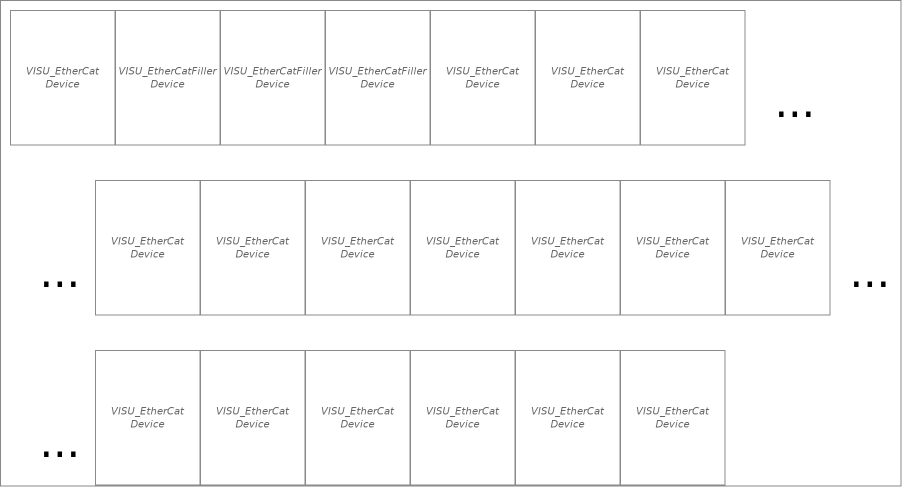
VISUALIZATION VISU_M1M2IO  // 902x487
VAR_IN_OUT
	ref : M1M2IO;
    widget : M1M2IOWidget;
END_VAR
    Frame (10,10 105x135)
        shows VISU_EtherCatDevice(device := ref.parts.COU, widget := widget.COU)
    Frame (535,10 105x135)
        shows VISU_EtherCatDevice(device := ref.parts.AI2, widget := widget.AI2)
    Frame (515,180 105x135)
        shows VISU_EtherCatDevice(device := ref.parts.RES3, widget := widget.RES3)
    Frame (640,10 105x135)
        shows VISU_EtherCatDevice(device := ref.parts.AI3, widget := widget.AI3)
    Frame (620,180 105x135)
        shows VISU_EtherCatDevice(device := ref.parts.PWR1, widget := widget.PWR1)
    Frame (95,180 105x135)
        shows VISU_EtherCatDevice(device := ref.parts.AO1, widget := widget.AO1)
    Frame (725,180 105x135)
        shows VISU_EtherCatDevice(device := ref.parts.SSI1, widget := widget.SSI1)
    Frame (200,180 105x135)
        shows VISU_EtherCatDevice(device := ref.parts.DO1, widget := widget.DO1)
    Frame (305,180 105x135)
        shows VISU_EtherCatDevice(device := ref.parts.RES1, widget := widget.RES1)
    Frame (410,180 105x135)
        shows VISU_EtherCatDevice(device := ref.parts.RES2, widget := widget.RES2)
    Frame (115,10 105x135)
        shows VISU_EtherCatFillerDevice()
    Frame (220,10 105x135)
        shows VISU_EtherCatFillerDevice()
    Frame (325,10 105x135)
        shows VISU_EtherCatFillerDevice()
    Label (765,70 60x64), "..."
    Label (30,240 60x64), "..."
    Frame (430,10 105x135)
        shows VISU_EtherCatDevice(device := ref.parts.AI1, widget := widget.AI1)
    Frame (410,350 105x135)
        shows VISU_EtherCatDevice(device := ref.parts.DO2, widget := widget.DO2)
    Frame (515,350 105x135)
        shows VISU_EtherCatDevice(device := ref.parts.DO3, widget := widget.DO3)
    Frame (95,350 105x135)
        shows VISU_EtherCatDevice(device := ref.parts.AI4, widget := widget.AI4)
    Frame (620,350 105x135)
        shows VISU_EtherCatDevice(device := ref.parts.RE1, widget := widget.RE1)
    Frame (200,350 105x135)
        shows VISU_EtherCatDevice(device := ref.parts.INC1, widget := widget.INC1)
    Frame (305,350 105x135)
        shows VISU_EtherCatDevice(device := ref.parts.P5V1, widget := widget.P5V1)
    Label (30,410 60x64), "..."
    Label (840,240 60x64), "..."
END_VISUALIZATION

(* stored: Version 1.1.0.1, ProductVersion 3.1.4019.2
   Visu VISU_M1M2IO: Id {fdca1858-9eb0-47dc-98cb-c124f4db3e9c} *)
